Fanuc KAREL source: kc00059.KL

-- PROVISIONAL review KL for V1013-1; original PC SHA256 8cd18822df23fd5952ce1f75da70fcd18d02f1f658b31350a54b0e932a90b636
-- Incomplete behavior may be omitted. Consult companion uncertainty JSON. Do not deploy.
PROGRAM KC00059
%NOLOCKGROUP
BEGIN
  -- UNRESOLVED_PC offsets 5-25; opcodes 27,27,9D,27,9D,22,AA,23
  -- UNRESOLVED_PC offsets 30-34; opcodes 7F
END KC00059
